{attribute 'qualified_only'}
VAR_GLOBAL
	HardwareInput		AT %I* : ARRAY [1..4] OF BOOL;
	HardwareOutput		AT %Q* : ARRAY [1..4] OF BOOL;
END_VAR

(* stored: Version 1.1.0.1, ProductVersion 3.1.4024.12
   GVL IO: Id {b4400bfc-3eb0-49f1-8284-15ad04357a14} *)
